Fanuc KAREL source: kt00523.KL

-- PROVISIONAL review KL for V1013-1; original PC SHA256 6f38275d71ec32273f944a7bdb3caf79cd7df66d8e3f98c2c076fbf70397f1e4
-- Incomplete behavior may be omitted. Consult companion uncertainty JSON. Do not deploy.
PROGRAM KT00523
%NOLOCKGROUP
VAR
  OUT : BOOLEAN
-- UNRESOLVED_DECL P1 type=000106
-- UNRESOLVED_DECL P2 type=000106
BEGIN
  -- UNRESOLVED_PC offsets 5-20; opcodes 2E,22,32,35
  -- UNRESOLVED_PC offsets 25-40; opcodes 2E,22,32,35
  -- UNRESOLVED_PC offsets 45-60; opcodes 2E,22,32,35
  -- UNRESOLVED_PC offsets 65-80; opcodes 2E,22,32,35
  -- UNRESOLVED_PC offsets 85-118; opcodes 49,7E,49,7E,AC,23
  -- UNRESOLVED_PC offsets 123-127; opcodes 7F
END KT00523
